TYPE ST_PeakshaveBox_Set :
STRUCT
	b_ContactorClose : BOOL;
	b_Alarm			 : BOOL;
	b_ExtIO			 : BOOL;
	b_BreakerControl : BOOL;
	ui_CtRange		 : UINT := 1000;
	r_VTRatio		 : REAL := 1;
	b_InverseCTdirection: BOOL;
END_STRUCT
END_TYPE

(* stored: Version 1.1.0.1, ProductVersion 3.1.4024.12
   DUT ST_PeakshaveBox_Set: Id {4978bb3b-3bd6-4034-a72d-1e677220775b} *)
